// TIA Portal project "Biegewerkzeug_2" (V20)

(* hardware
DEVICE "S7-1500/ET200MP-Station_1"  S7-1500 station
   slot 0: "Profilschiene_0"  Rack  6ES7 590-1***0-0AA0
   slot 1: "PLC_1"  CPU 1513-1 PN  6ES7 513-1AM03-0AB0  V4.0
      slot 3: "CPU-Display_1"  6ES7591-1AA00-0AA0
      slot 32768: "PROFINET-Schnittstelle_1"  X1
         slot 32769: "Port_1"  X1 P1
         slot 32770: "Port_2"  X1 P2
      slot 34817: "Virtual CP interface port_1"  Virtual CP interface port  Virtual CP interface port FW V4.0
   slot 2: "DI 16x24VDC BA_1"  DI 16x24VDC BA  6ES7 521-1BH10-0AA0  V1.1
   slot 3: "DQ 16x24VDC/0.5A ST_1"  DQ 16x24VDC/0.5A ST  6ES7 522-1BH00-0AB0  V2.0
   slot 4: "AI 8xU/I/R/RTD BA_2"  AI 8xU/I/R/RTD BA  6ES7 531-7QF00-0AB0  V1.0
   slot 5: "AQ 8xU/I HS_2"  AQ 8xU/I HS  6ES7 532-5HF00-0AB0  V2.2
*)

// ===== PLC "PLC_1"  CPU 1513-1 PN =====

VAR_GLOBAL   // PLC tag table "Standard-Variablentabelle"
   "Clock_Byte" AT %MB0 : Byte;
   "Clock_10Hz" AT %M0.0 : Bool;
   "Clock_5Hz" AT %M0.1 : Bool;
   "Clock_2.5Hz" AT %M0.2 : Bool;
   "Clock_2Hz" AT %M0.3 : Bool;
   "Clock_1.25Hz" AT %M0.4 : Bool;
   "Clock_1Hz" AT %M0.5 : Bool;
   "Clock_0.625Hz" AT %M0.6 : Bool;
   "Clock_0.5Hz" AT %M0.7 : Bool;
END_VAR

VAR_GLOBAL   // PLC tag table "Eingaenge"
   "S1" AT %I0.0 : Bool;   // Starttaster
   "1B1" AT %I0.1 : Bool;   // Kolben_1 - Sensor hinten
   "1B2" AT %I0.2 : Bool;   // Kolben_1 - Sensor vorne
   "2B1" AT %I0.3 : Bool;   // Kolben_2 - Sensor hinten
   "2B2" AT %I0.4 : Bool;   // Kolben_2 - Sensor vorne
   "S3" AT %E1.2 : Bool;   // Starttaster
   "S2" AT %E0.5 : Bool;   // Starttaster
   "5B1" AT %E1.3 : Bool;   // Kolben_1 - Sensor hinten
   "3B1" AT %E0.6 : Bool;   // Kolben_1 - Sensor hinten
   "5B2" AT %E1.4 : Bool;   // Kolben_1 - Sensor vorne
   "3B2" AT %E0.7 : Bool;   // Kolben_1 - Sensor vorne
   "6B1" AT %E1.5 : Bool;   // Kolben_2 - Sensor hinten
   "4B1" AT %E1.0 : Bool;   // Kolben_2 - Sensor hinten
   "6B2" AT %E1.6 : Bool;   // Kolben_2 - Sensor vorne
   "4B2" AT %E1.1 : Bool;   // Kolben_2 - Sensor vorne
END_VAR

VAR_GLOBAL   // PLC tag table "Ausgaenge"
   "H1" AT %Q0.0 : Bool;   // Startleuchte
   "1M1" AT %Q0.1 : Bool;   // Kolben_1 - Motor
   "2M1" AT %Q0.3 : Bool;   // Kolben_2 - Motor
   "H3" AT %A1.2 : Bool;   // Startleuchte
   "H2" AT %A0.5 : Bool;   // Startleuchte
   "5M1" AT %A1.3 : Bool;   // Kolben_1 - Motor
   "3M1" AT %A0.6 : Bool;   // Kolben_1 - Motor
   "6M1" AT %A1.5 : Bool;   // Kolben_2 - Motor
   "4M1" AT %A1.0 : Bool;   // Kolben_2 - Motor
   "Prozessstart" AT %E1.7 : Bool;
END_VAR

DATA_BLOCK "Biegeprozess_DB_1"   // DB1
{ S7_Optimized_Access := 'TRUE' }
VERSION : 0.1
// stored: InstanceOfName Biegeprozess
"Biegeprozess"
BEGIN
END_DATA_BLOCK

DATA_BLOCK "Biegeprozess_DB_2"   // DB2
{ S7_Optimized_Access := 'TRUE' }
VERSION : 0.1
// stored: InstanceOfName Biegeprozess
"Biegeprozess"
BEGIN
END_DATA_BLOCK

DATA_BLOCK "Biegeprozess_DB_3"   // DB3
{ S7_Optimized_Access := 'TRUE' }
VERSION : 0.1
// stored: InstanceOfName Biegeprozess
"Biegeprozess"
BEGIN
END_DATA_BLOCK

DATA_BLOCK "DB_1"   // DB6
{ S7_Optimized_Access := 'TRUE' }
VERSION : 0.1
   VAR
      IEC_Zaehler : Array[0..2] of IEC_DCOUNTER;
   END_VAR
BEGIN
END_DATA_BLOCK

FUNCTION_BLOCK "Biegeprozess"   // FB1, FBD
{ S7_Optimized_Access := 'TRUE' }
VERSION : 0.1
   VAR_INPUT
      Prozessstart : Bool;
      Sensor_1_hinten : Bool;
      Sensor_1_vorne : Bool;
      Sensor_2_hinten : Bool;
      Sensor_2_vorne : Bool;
   END_VAR
   VAR_OUTPUT
      Motor_1_Kolben : Bool;
      Motor_2_Kolben : Bool;
      Melde_Leuchte : Bool;
   END_VAR
   VAR_IN_OUT
      Schritt_Zaehler : IEC_DCOUNTER;
   END_VAR
   VAR
      Prozessschritte : Struct
         Schritt : Struct
            "1_starten" : Bool;
            "1_beendet" : Bool;
            "2_starten" : Bool;
            "2_beendet" : Bool;
         END_STRUCT;
         Prozessende : Bool := True;
         Zaehler : DInt;
      END_STRUCT;
   END_VAR
BEGIN

REGION Network 1
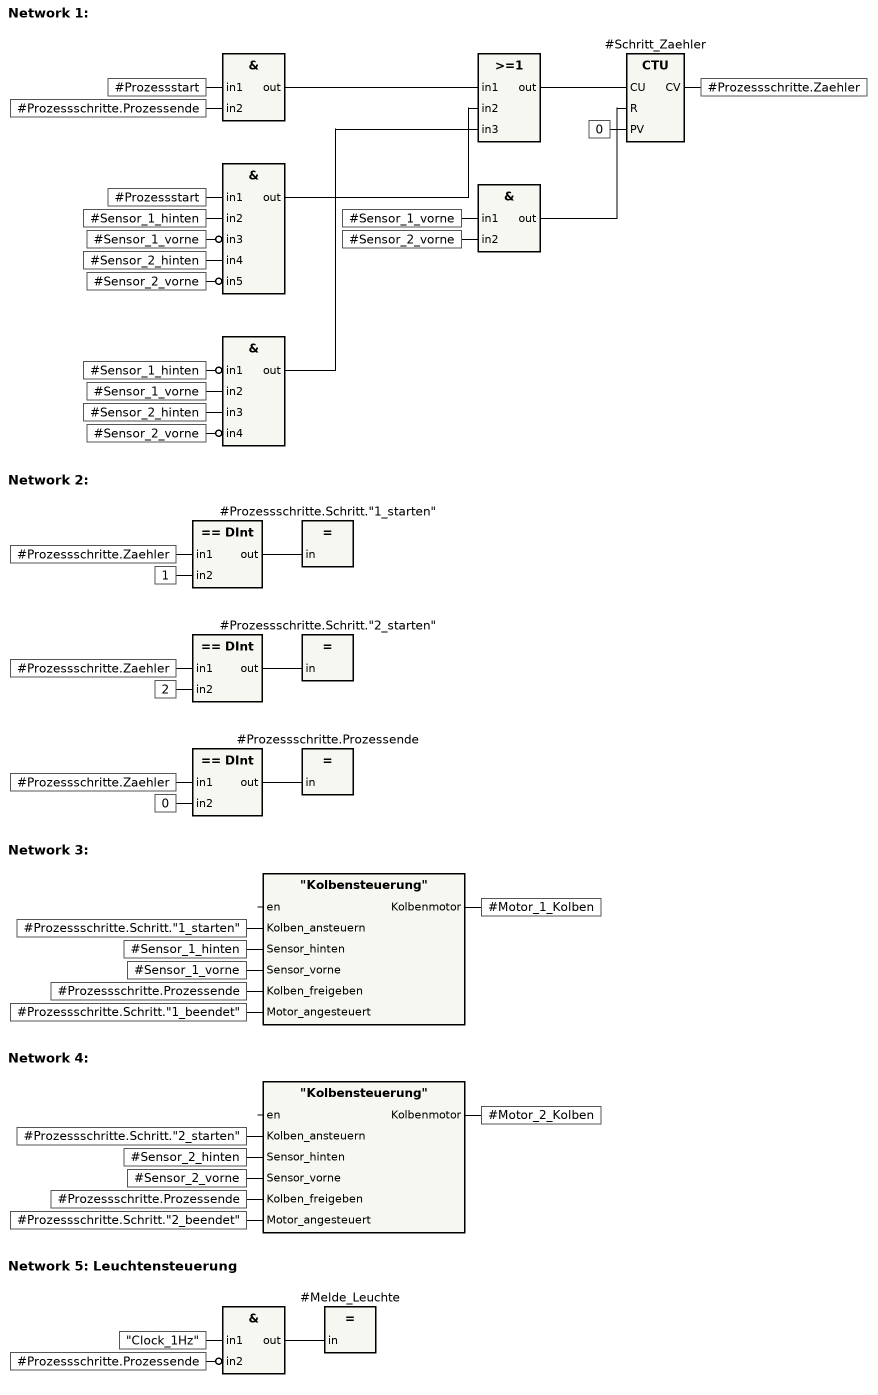
   #Schritt_Zaehler.CTU(CU := (#Prozessstart AND #Prozessschritte.Prozessende) OR (#Prozessstart AND #Sensor_1_hinten AND NOT #Sensor_1_vorne AND #Sensor_2_hinten AND NOT #Sensor_2_vorne) OR (NOT #Sensor_1_hinten AND #Sensor_1_vorne AND #Sensor_2_hinten AND NOT #Sensor_2_vorne),
                        R := #Sensor_1_vorne AND #Sensor_2_vorne,
                        PV := 0,
                        CV => #Prozessschritte.Zaehler);
END_REGION

REGION Network 2
   #Prozessschritte.Schritt."1_starten" := #Prozessschritte.Zaehler = 1;
   #Prozessschritte.Schritt."2_starten" := #Prozessschritte.Zaehler = 2;
   #Prozessschritte.Prozessende := #Prozessschritte.Zaehler = 0;
END_REGION

REGION Network 3
   "Kolbensteuerung"(Kolben_ansteuern := #Prozessschritte.Schritt."1_starten",
                     Sensor_hinten := #Sensor_1_hinten,
                     Sensor_vorne := #Sensor_1_vorne,
                     Kolben_freigeben := #Prozessschritte.Prozessende,
                     Motor_angesteuert := #Prozessschritte.Schritt."1_beendet",
                     Kolbenmotor => #Motor_1_Kolben);
END_REGION

REGION Network 4
   "Kolbensteuerung"(Kolben_ansteuern := #Prozessschritte.Schritt."2_starten",
                     Sensor_hinten := #Sensor_2_hinten,
                     Sensor_vorne := #Sensor_2_vorne,
                     Kolben_freigeben := #Prozessschritte.Prozessende,
                     Motor_angesteuert := #Prozessschritte.Schritt."2_beendet",
                     Kolbenmotor => #Motor_2_Kolben);
END_REGION

REGION Network 5: Leuchtensteuerung
   #Melde_Leuchte := "Clock_1Hz" AND NOT #Prozessschritte.Prozessende;
END_REGION
END_FUNCTION_BLOCK

FUNCTION "Kolbensteuerung" : Void   // FC1, FBD
{ S7_Optimized_Access := 'TRUE' }
VERSION : 0.1
   VAR_INPUT
      Kolben_ansteuern : Bool;
      Sensor_hinten : Bool;
      Sensor_vorne : Bool;
   END_VAR
   VAR_OUTPUT
      Kolbenmotor : Bool;
   END_VAR
   VAR_IN_OUT
      Kolben_freigeben : Bool;
      Motor_angesteuert : Bool;
   END_VAR
BEGIN

REGION Network 1
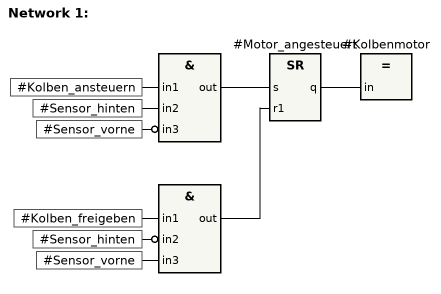
   IF #Kolben_ansteuern AND #Sensor_hinten AND NOT #Sensor_vorne THEN
       #Motor_angesteuert := TRUE;   // SR flip-flop
   END_IF;
   IF #Kolben_freigeben AND NOT #Sensor_hinten AND #Sensor_vorne THEN #Motor_angesteuert := FALSE; END_IF;
   #Kolbenmotor := #Motor_angesteuert;
END_REGION
END_FUNCTION

ORGANIZATION_BLOCK "Main"   // OB1, FBD, ProgramCycle
TITLE = "Main Program Sweep (Cycle)"
{ S7_Optimized_Access := 'TRUE' }
VERSION : 0.1
   VAR_INPUT
      Initial_Call : Bool;   // Initial call of this OB
      Remanence : Bool;   // =True, if remanent data are available
   END_VAR
BEGIN

REGION Network 1
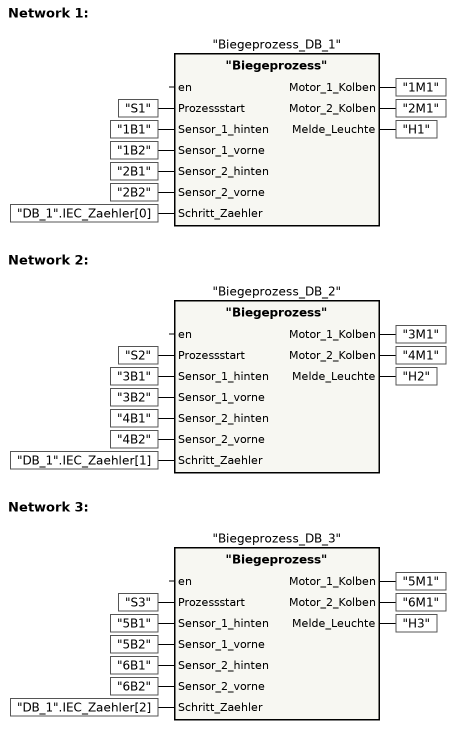
   "Biegeprozess_DB_1"(Prozessstart := "S1",   // "Biegeprozess"
                       Sensor_1_hinten := "1B1",
                       Sensor_1_vorne := "1B2",
                       Sensor_2_hinten := "2B1",
                       Sensor_2_vorne := "2B2",
                       Schritt_Zaehler := "DB_1".IEC_Zaehler[0],
                       Motor_1_Kolben => "1M1",
                       Motor_2_Kolben => "2M1",
                       Melde_Leuchte => "H1");
END_REGION

REGION Network 2
   "Biegeprozess_DB_2"(Prozessstart := "S2",   // "Biegeprozess"
                       Sensor_1_hinten := "3B1",
                       Sensor_1_vorne := "3B2",
                       Sensor_2_hinten := "4B1",
                       Sensor_2_vorne := "4B2",
                       Schritt_Zaehler := "DB_1".IEC_Zaehler[1],
                       Motor_1_Kolben => "3M1",
                       Motor_2_Kolben => "4M1",
                       Melde_Leuchte => "H2");
END_REGION

REGION Network 3
   "Biegeprozess_DB_3"(Prozessstart := "S3",   // "Biegeprozess"
                       Sensor_1_hinten := "5B1",
                       Sensor_1_vorne := "5B2",
                       Sensor_2_hinten := "6B1",
                       Sensor_2_vorne := "6B2",
                       Schritt_Zaehler := "DB_1".IEC_Zaehler[2],
                       Motor_1_Kolben => "5M1",
                       Motor_2_Kolben => "6M1",
                       Melde_Leuchte => "H3");
END_REGION
END_ORGANIZATION_BLOCK